// TIA Portal project "2022.04.23-三色报警灯" (V17)

(* hardware
DEVICE "S7-1500/ET200MP station_1"  S7-1500 station
   slot 0: "导轨_0"  Rack  6ES7 590-1***0-0AA0
   slot 1: "PLC_1"  CPU 1516-3 PN/DP  6ES7 516-3AN00-0AB0  V1.7
      slot 3: "CPU 显示_1"  6ES7591-1BA00-0AA0
      slot 32768: "PROFINET 接口_1"  X1
         slot 32769: "端口_1"  X1 P1
         slot 32770: "端口_2"  X1 P2
      slot 33024: "PROFINET 接口_2"  X2
         slot 33025: "端口_1"  X2 P1
      slot 33280: "DP 接口_1"  X3
   slot 2: "DI 32x24VDC BA_1"  DI 32x24VDC BA  6ES7 521-1BL10-0AA0  V1.1
   slot 3: "DQ 32x24VDC/0.5A HF_1"  DQ 32x24VDC/0.5A HF  6ES7 522-1BL01-0AB0  V1.1
*)

// ===== PLC "PLC_1"  CPU 1516-3 PN/DP =====

VAR_GLOBAL   // PLC tag table "默认变量表"
   "跳闸报警" AT %I0.0 : Bool;
   "堵塞报警" AT %I0.1 : Bool;
   "超时报警" AT %I0.2 : Bool;
   "复位按钮" AT %I0.3 : Bool;
   "按钮5" AT %I0.4 : Bool;
   "按钮6" AT %I0.5 : Bool;
   "按钮7" AT %I0.6 : Bool;
   "按钮8" AT %I0.7 : Bool;
   "按钮9" AT %I1.0 : Bool;
   "按钮10" AT %I1.1 : Bool;
   "按钮11" AT %I1.2 : Bool;
   "自动指示灯" AT %Q0.0 : Bool;
   "手动指示灯" AT %Q0.1 : Bool;
   "故障指示灯" AT %Q0.2 : Bool;
   "蜂鸣器" AT %Q0.3 : Bool;
   "指示灯5" AT %Q0.4 : Bool;
   "指示灯6" AT %Q0.5 : Bool;
   "指示灯7" AT %Q0.6 : Bool;
   "指示灯8" AT %Q0.7 : Bool;
   "指示灯9" AT %Q1.0 : Bool;
   "指示灯10" AT %Q1.1 : Bool;
   "指示灯11" AT %Q1.2 : Bool;
   "指示灯12" AT %Q1.3 : Bool;
   "System_Byte" AT %MB0 : Byte;
   "FirstScan" AT %M0.0 : Bool;
   "DiagStatusUpdate" AT %M0.1 : Bool;
   "AlwaysTRUE" AT %M0.2 : Bool;
   "AlwaysFALSE" AT %M0.3 : Bool;
   "Clock_Byte" AT %MB0 : Byte;
   "Clock_10Hz" AT %M0.0 : Bool;
   "Clock_5Hz" AT %M0.1 : Bool;
   "Clock_2.5Hz" AT %M0.2 : Bool;
   "Clock_2Hz" AT %M0.3 : Bool;
   "Clock_1.25Hz" AT %M0.4 : Bool;
   "Clock_1Hz" AT %M0.5 : Bool;
   "Clock_0.625Hz" AT %M0.6 : Bool;
   "Clock_0.5Hz" AT %M0.7 : Bool;
   "手/自切换" AT %M1.0 : Bool;
   "报警状态" AT %M1.1 : Bool;
END_VAR

FUNCTION "报警LAD" : Void   // FC1, LAD
{ S7_Optimized_Access := 'TRUE' }
VERSION : 0.1
BEGIN

REGION Network 1: 自动状态
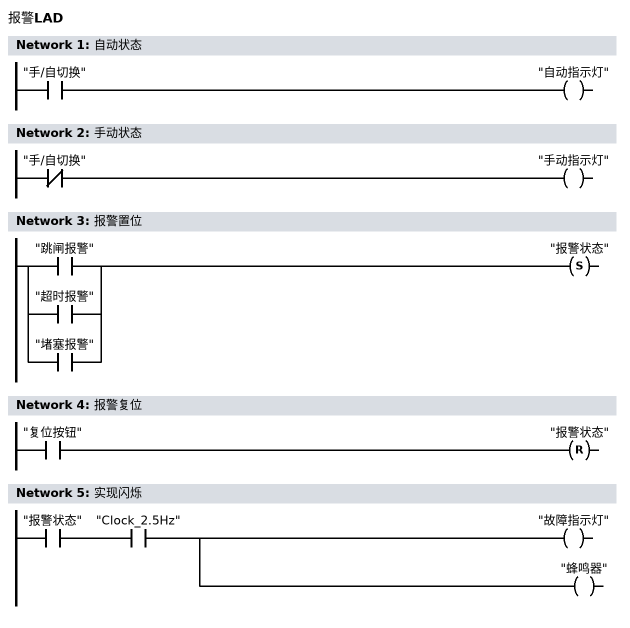
   RUNG wire#powerrail
      Contact( "手/自切换" )
      Coil( "自动指示灯" )
   END_RUNG
   // the same network as SCL:
   "自动指示灯" := "手/自切换";
END_REGION

REGION Network 2: 手动状态
   RUNG wire#powerrail
      I_Contact( "手/自切换" )
      Coil( "手动指示灯" )
   END_RUNG
   // the same network as SCL:
   "手动指示灯" := NOT "手/自切换";
END_REGION

REGION Network 3: 报警置位
   RUNG wire#powerrail
      Contact( "跳闸报警" )
      wire#w1
      S_Coil( "报警状态" )
   END_RUNG
   RUNG wire#powerrail
      Contact( "超时报警" )
   END_RUNG wire#w1
   RUNG wire#powerrail
      Contact( "堵塞报警" )
   END_RUNG wire#w1
   // the same network as SCL:
   IF "跳闸报警" OR "超时报警" OR "堵塞报警" THEN "报警状态" := TRUE; END_IF;
END_REGION

REGION Network 4: 报警复位
   RUNG wire#powerrail
      Contact( "复位按钮" )
      R_Coil( "报警状态" )
   END_RUNG
   // the same network as SCL:
   IF "复位按钮" THEN "报警状态" := FALSE; END_IF;
END_REGION

REGION Network 5: 实现闪烁
   RUNG wire#powerrail
      Contact( "报警状态" )
      Contact( "Clock_2.5Hz" )
      wire#w1
      Coil( "故障指示灯" )
   END_RUNG
   RUNG wire#w1
      Coil( "蜂鸣器" )
   END_RUNG
   // the same network as SCL:
   "故障指示灯" := "报警状态" AND "Clock_2.5Hz";
   "蜂鸣器" := "故障指示灯";
END_REGION
END_FUNCTION

FUNCTION "报警FBD" : Void   // FC2, FBD
{ S7_Optimized_Access := 'TRUE' }
VERSION : 0.1
BEGIN

REGION Network 1: 手自动状态
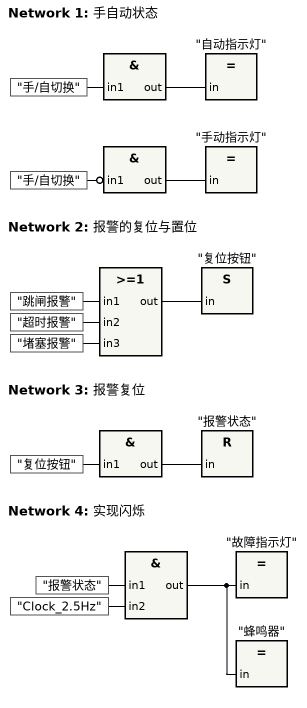
   "自动指示灯" := "手/自切换";
   "手动指示灯" := NOT "手/自切换";
END_REGION

REGION Network 2: 报警的复位与置位
   IF "跳闸报警" OR "超时报警" OR "堵塞报警" THEN "复位按钮" := TRUE; END_IF;
END_REGION

REGION Network 3: 报警复位
   IF "复位按钮" THEN "报警状态" := FALSE; END_IF;
END_REGION

REGION Network 4: 实现闪烁
   "故障指示灯" := "报警状态" AND "Clock_2.5Hz";
   "蜂鸣器" := "故障指示灯";
END_REGION
END_FUNCTION

FUNCTION "报警SCL" : Void   // FC3, SCL
{ S7_Optimized_Access := 'TRUE' }
VERSION : 0.1
BEGIN
   //手自动状态
   IF "手/自切换" THEN
       "自动指示灯" := 1;
       "手动指示灯" := 0
       ;
   ELSE
       "自动指示灯" := 0;
       "手动指示灯" := 1
       ;
   END_IF;

   //报警复位
   IF "跳闸报警" OR "超时报警" OR "堵塞报警" THEN
       "报警状态" := TRUE;
   END_IF;
   //报警复位
   IF "复位按钮" THEN
       "报警状态" := FALSE;
   END_IF;
       //实现报警闪烁
   IF "报警状态" & "Clock_2.5Hz" THEN
       "故障指示灯" := 1;

       "蜂鸣器" := 1;
   ELSE
       "故障指示灯" := 0;

       "蜂鸣器" := 0;
   END_IF;
END_FUNCTION

ORGANIZATION_BLOCK "Main"   // OB1, LAD, ProgramCycle
TITLE = "Main Program Sweep (Cycle)"
{ S7_Optimized_Access := 'TRUE' }
VERSION : 0.1
   VAR_INPUT
      Initial_Call : Bool;   // Initial call of this OB
      Remanence : Bool;   // =True, if remanent data are available
   END_VAR
BEGIN

REGION Network 1: 1
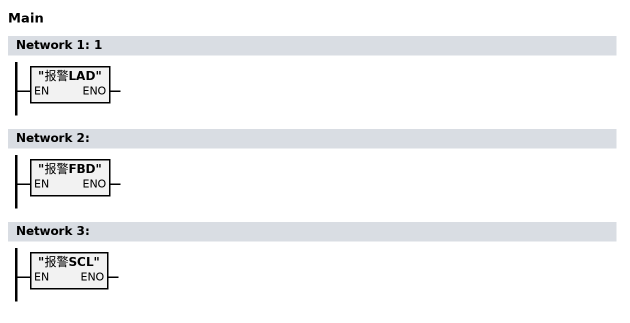
   RUNG wire#powerrail
      "报警LAD"()
   END_RUNG
   // the same network as SCL:
   "报警LAD"();
END_REGION

REGION Network 2
   RUNG wire#powerrail
      "报警FBD"()
   END_RUNG
   // the same network as SCL:
   "报警FBD"();
END_REGION

REGION Network 3
   RUNG wire#powerrail
      "报警SCL"()
   END_RUNG
   // the same network as SCL:
   "报警SCL"();
END_REGION
END_ORGANIZATION_BLOCK